FUNCTION_BLOCK Section2Ctrl
  (* Standard: 61499-2 *)
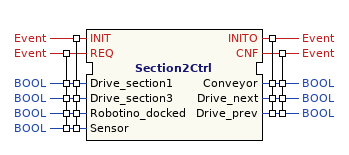
  EVENT_INPUT
    INIT WITH Drive_section1, Drive_section3, Robotino_docked, Sensor;
    REQ WITH Drive_section1, Drive_section3, Robotino_docked, Sensor;
  END_EVENT
  EVENT_OUTPUT
    INITO WITH Conveyor, Drive_next, Drive_prev;
    CNF WITH Conveyor, Drive_next, Drive_prev;
  END_EVENT
  VAR_INPUT
    Drive_section1 : BOOL;
    Drive_section3 : BOOL;
    Robotino_docked : BOOL;
    Sensor : BOOL;
  END_VAR
  VAR_OUTPUT
    Conveyor : BOOL;
    Drive_next : BOOL;
    Drive_prev : BOOL;
  END_VAR
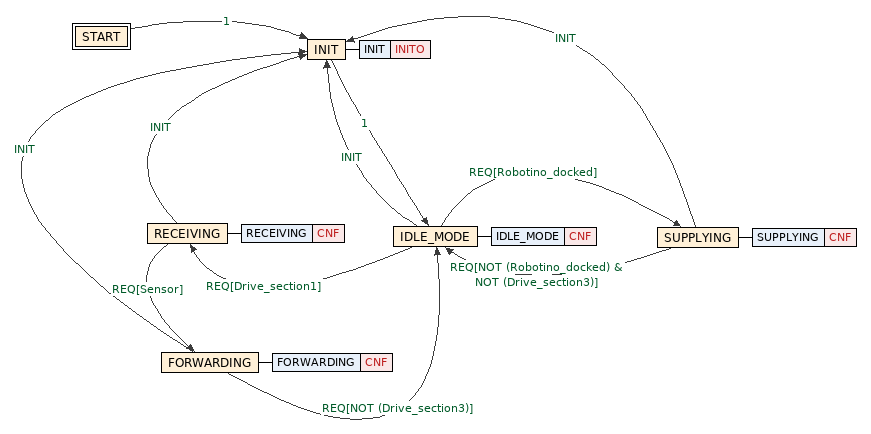
  EC_STATES
    START;
    INIT : INIT -> INITO;
    IDLE_MODE : IDLE_MODE -> CNF;
    SUPPLYING : SUPPLYING -> CNF;
    RECEIVING : RECEIVING -> CNF;
    FORWARDING : FORWARDING -> CNF;
  END_STATES
  EC_TRANSITIONS
    START TO INIT := 1;
    INIT TO IDLE_MODE := 1;
    IDLE_MODE TO SUPPLYING := REQ[Robotino_docked];
    SUPPLYING TO IDLE_MODE := REQ[NOT (Robotino_docked) & NOT (Drive_section3)];
    IDLE_MODE TO RECEIVING := REQ[Drive_section1];
    RECEIVING TO FORWARDING := REQ[Sensor];
    FORWARDING TO IDLE_MODE := REQ[NOT (Drive_section3)];
    IDLE_MODE TO INIT := INIT;
    SUPPLYING TO INIT := INIT;
    FORWARDING TO INIT := INIT;
    RECEIVING TO INIT := INIT;
  END_TRANSITIONS
  ALGORITHM INIT IN ST:
Conveyor := FALSE;&#10;Drive_next := FALSE;&#10;Drive_prev := FALSE;&#10;
  END_ALGORITHM
  ALGORITHM REQ IN ST:

  END_ALGORITHM
  ALGORITHM IDLE_MODE IN ST:
Conveyor := FALSE;&#10;Drive_next := FALSE;&#10;Drive_prev := TRUE;&#10;
  END_ALGORITHM
  ALGORITHM SUPPLYING IN ST:
Conveyor := TRUE;&#10;Drive_next := TRUE;&#10;Drive_prev := FALSE;&#10;
  END_ALGORITHM
  ALGORITHM RECEIVING IN ST:
Conveyor := TRUE;&#10;Drive_next := FALSE;&#10;Drive_prev := TRUE;&#10;
  END_ALGORITHM
  ALGORITHM FORWARDING IN ST:
Conveyor := TRUE;&#10;Drive_next := TRUE;&#10;Drive_prev := FALSE;&#10;
  END_ALGORITHM
END_FUNCTION_BLOCK
